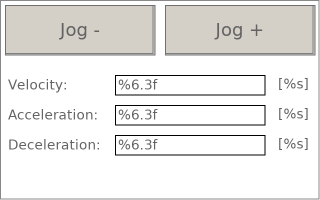
VISUALIZATION SingleAxisJogContinous  // 320x200
VAR_IN_OUT
	btnJogPositive	: BOOL;
	btnJogNegative	: BOOL;
	lrVelocity		: LREAL;
	lrAcceleration	: LREAL;
	lrDeceleration	: LREAL;
	sUnit			: STRING;
END_VAR
    Rectangle (5,75 110x20), "Velocity:"
    Rectangle (115,75 150x20), "%6.3f", text variable: lrVelocity
        OnMouseClick: write the text variable via VisuDialogs.Numpad
    Rectangle (275,75 44x18), "[%s]", text variable: sUnit
    Button (5,5 150x50), "Jog -"
        tap btnJogNegative
        OnMouseUp: toggle btnJogNegative
        OnMouseDown: toggle btnJogNegative
    Button (165,5 150x50), "Jog +"
        tap btnJogPositive
    Rectangle (5,105 110x20), "Acceleration:"
    Rectangle (115,105 150x20), "%6.3f", text variable: lrAcceleration
        OnMouseClick: write the text variable via VisuDialogs.Numpad
    Rectangle (275,105 44x18), "[%s]", text variable: sUnit
    Rectangle (5,135 110x20), "Deceleration:"
    Rectangle (115,135 150x20), "%6.3f", text variable: lrDeceleration
        OnMouseClick: write the text variable via VisuDialogs.Numpad
    Rectangle (275,135 44x18), "[%s]", text variable: sUnit
END_VISUALIZATION

(* stored: Version 1.1.0.1, ProductVersion 3.1.4024.9
   Visu SingleAxisJogContinous: Id {02371741-e252-40b5-b156-605ccb4c6be5} *)
